(* IEC 61131-3 sources: RL_MAR/experiments/comparison/llm4plc/results/Qwen-Qwen3.5-9B_20260506_150728/20260506_170107, 4 files *)

(* ---- generated_code_iteration_0.st ---- *)
START_ST
FUNCTION_BLOCK PouchMachine
VAR_INPUT
    start_machine: BOOL;
    stop_machine: BOOL;
END_VAR

VAR_OUTPUT
    machine_ready: BOOL;
    feeder_running: BOOL;
    cutter_running: BOOL;
    heating_running: BOOL;
    cooling_running: BOOL;
END_VAR

VAR
    current_state: INT;
    prev_state: INT;

    station_heating_ready: ARRAY[0..7] OF BOOL;
    station_cooling_ready: ARRAY[0..7] OF BOOL;
    tension_stable: BOOL;
    cutter_h_stopped: BOOL;
    cutter_v_stopped: BOOL;
    feeder_1_stopped: BOOL;
    feeder_2_stopped: BOOL;

    ctrl_heating: BOOL;
    ctrl_cooling: BOOL;
    ctrl_feeders: BOOL;
    ctrl_cutters: BOOL;
END_VAR

END_VAR

BEGIN
    (* STATE 0: IDLE *)
    IF current_state = 0 THEN
        machine_ready := FALSE;
        feeder_running := FALSE;
        cutter_running := FALSE;
        heating_running := FALSE;
        cooling_running := FALSE;

        (* Transition to STATE 1 *)
        IF start_machine = TRUE AND stop_machine = FALSE THEN
            current_state := 1;
        END_IF;
    END_IF;

    (* STATE 1: INITIATE_STARTUP *)
    IF current_state = 1 THEN
        machine_ready := FALSE;
        feeder_running := FALSE;
        cutter_running := FALSE;
        heating_running := FALSE;
        cooling_running := FALSE;

        (* Check if all heating and cooling stations are ready to proceed to warmup *)
        IF start_machine = TRUE AND stop_machine = FALSE THEN
            heating_running := TRUE;
            cooling_running := TRUE;
            ctrl_heating := TRUE;
            ctrl_cooling := TRUE;
            ctrl_feeders := FALSE;
            ctrl_cutters := FALSE;

            (* Check if all stations report ready to move to STATE 2 (Warmup Active) *)
            (* Note: Logic assumes 'ready' implies active heating/cooling cycle start *)
            IF (station_heating_ready[0] AND station_heating_ready[1] AND station_heating_ready[2] AND station_heating_ready[3] AND
                station_heating_ready[4] AND station_heating_ready[5] AND station_heating_ready[6] AND station_heating_ready[7]) AND
               (station_cooling_ready[0] AND station_cooling_ready[1] AND station_cooling_ready[2] AND station_cooling_ready[3] AND
                station_cooling_ready[4] AND station_cooling_ready[5] AND station_cooling_ready[6] AND station_cooling_ready[7]) THEN
                current_state := 2;
            END_IF;
        END_IF;
    END_IF;

    (* STATE 2: WARMUP_STATIONS *)
    IF current_state = 2 THEN
        machine_ready := FALSE;
        feeder_running := FALSE;
        cutter_running := FALSE;
        heating_running := TRUE;
        cooling_running := TRUE;

        (* Logic: Wait until all stations report "Ready/Active" to move to STATE 3 *)
        (* In this context, we assume the 'ready' flag indicates the warmup cycle is complete and stable *)
        IF start_machine = TRUE AND stop_machine = FALSE THEN
            IF (station_heating_ready[0] AND station_heating_ready[1] AND station_heating_ready[2] AND station_heating_ready[3] AND
                station_heating_ready[4] AND station_heating_ready[5] AND station_heating_ready[6] AND station_heating_ready[7]) AND
               (station_cooling_ready[0] AND station_cooling_ready[1] AND station_cooling_ready[2] AND station_cooling_ready[3] AND
                station_cooling_ready[4] AND station_cooling_ready[5] AND station_cooling_ready[6] AND station_cooling_ready[7]) THEN
                current_state := 3;
            END_IF;
        END_IF;
    END_IF;

    (* STATE 3: TENSION_ESTABLISHMENT *)
    IF current_state = 3 THEN
        machine_ready := FALSE;
        feeder_running := TRUE;
        cutter_running := FALSE;
        heating_running := TRUE;
        cooling_running := TRUE;

        ctrl_heating := TRUE;
        ctrl_cooling := TRUE;
        ctrl_feeders := TRUE;
        ctrl_cutters := FALSE;

        (* Logic: Monitor tension sensor. Once tension is stable, move to STATE 4 *)
        IF start_machine = TRUE AND stop_machine = FALSE AND tension_stable = TRUE THEN
            current_state := 4;
        END_IF;
    END_IF;

    (* STATE 4: OPERATIONAL_READY *)
    IF current_state = 4 THEN
        machine_ready := TRUE;
        feeder_running := TRUE;
        cutter_running := FALSE;
        heating_running := TRUE;
        cooling_running := TRUE;

        ctrl_heating := TRUE;
        ctrl_cooling := TRUE;
        ctrl_feeders := TRUE;
        ctrl_cutters := FALSE;

        (* Logic: Wait for stop_machine signal to move to STATE 5 *)
        IF stop_machine = TRUE THEN
            current_state := 5;
        END_IF;
    END_IF;

    (* STATE 5: INITIATE_SHUTDOWN *)
    IF current_state = 5 THEN
        machine_ready := FALSE;
        feeder_running := TRUE;
        cutter_running := FALSE;
        heating_running := TRUE;
        cooling_running := TRUE;

        ctrl_heating := TRUE;
        ctrl_cooling := TRUE;
        ctrl_feeders := TRUE;
        ctrl_cutters := FALSE;

        (* Logic: Immediately stop cutters to move to STATE 6 *)
        ctrl_cutters := FALSE;
        current_state := 6;
    END_IF;

    (* STATE 6: CUTTER_STOP *)
    IF current_state = 6 THEN
        machine_ready := FALSE;
        feeder_running := TRUE;
        cutter_running := FALSE;
        heating_running := TRUE;
        cooling_running := TRUE;

        ctrl_heating := TRUE;
        ctrl_cooling := TRUE;
        ctrl_feeders := TRUE;
        ctrl_cutters := FALSE;

        (* Logic: Wait until both cutters report "Stopped" to move to STATE 7 *)
        IF stop_machine = TRUE AND cutter_h_stopped = TRUE AND cutter_v_stopped = TRUE THEN
            current_state := 7;
        END_IF;
    END_IF;

    (* STATE 7: FEEDER_STOP *)
    IF current_state = 7 THEN
        machine_ready := FALSE;
        feeder_running := FALSE;
        cutter_running := FALSE;
        heating_running := TRUE;
        cooling_running := TRUE;

        ctrl_heating := TRUE;
        ctrl_cooling := TRUE;
        ctrl_feeders := FALSE;
        ctrl_cutters := FALSE;

        (* Logic: Wait until both feeders report "Stopped" to move to STATE 8 *)
        IF stop_machine = TRUE AND feeder_1_stopped = TRUE AND feeder_2_stopped = TRUE THEN
            current_state := 8;
        END_IF;
    END_IF;

    (* STATE 8: STATION_COOLDOWN *)
    IF current_state = 8 THEN
        machine_ready := FALSE;
        feeder_running := FALSE;
        cutter_running := FALSE;
        heating_running := FALSE;
        cooling_running := FALSE;

        ctrl_heating := FALSE;
        ctrl_cooling := FALSE;
        ctrl_feeders := FALSE;
        ctrl_cutters := FALSE;

        (* Logic: Wait until all heating/cooling stations report "Off/Inactive" to move to STATE 9 *)
        IF stop_machine = TRUE AND
           (station_heating_ready[0] = FALSE AND station_heating_ready[1] = FALSE AND station_heating_ready[2] = FALSE AND station_heating_ready[3] = FALSE AND
            station_heating_ready[4] = FALSE AND station_heating_ready[5] = FALSE AND station_heating_ready[6] = FALSE AND station_heating_ready[7] = FALSE) AND
           (station_cooling_ready[0] = FALSE AND station_cooling_ready[1] = FALSE AND station_cooling_ready[2] = FALSE AND station_cooling_ready[3] = FALSE AND
            station_cooling_ready[4] = FALSE AND station_cooling_ready[5] = FALSE AND station_cooling_ready[6] = FALSE AND station_cooling_ready[7] = FALSE) THEN
            current_state := 9;
        END_IF;
    END_IF;

    (* STATE 9: IDLE_RETURN *)
    IF current_state = 9 THEN
        machine_ready := FALSE;
        feeder_running := FALSE;
        cutter_running := FALSE;
        heating_running := FALSE;
        cooling_running := FALSE;

        ctrl_heating := FALSE;
        ctrl_cooling := FALSE;
        ctrl_feeders := FALSE;
        ctrl_cutters := FALSE;

        (* Logic: Remain here until start_machine is pressed again *)
        IF start_machine = TRUE THEN
            current_state := 1;
        END_IF;
    END_IF;

END_FUNCTION_BLOCK
END_ST

(* ---- generated_code_iteration_1.st ---- *)
START_REASON
The previous code failed CODESYS compiler validation (Error 500) primarily due to a structural syntax error in the `FUNCTION_BLOCK` definition. Specifically, the `END_VAR` keyword was placed immediately after the `VAR` section without a `END_VAR` closing the `VAR` block itself, or rather, the structure was malformed such that the compiler could not distinguish between the end of the variable list and the end of the block header.

In IEC 61131-3 Structured Text:
1. The `VAR` section must be closed with `END_VAR`.
2. The `FUNCTION_BLOCK` body (the `BEGIN...END` block) must be closed with `END_FUNCTION_BLOCK`.
3. The `END_VAR` seen in the original code after the `VAR` section was likely misplaced or the `VAR` section was not properly terminated before the `BEGIN` keyword, causing the parser to fail when it encountered the `BEGIN` or the subsequent `END_FUNCTION_BLOCK`.

Additionally, while not strictly causing the compile error, the logic for state transitions often benefits from initializing state variables at the start of the execution cycle to prevent undefined behavior on the first scan, though the primary fix required is the structural syntax correction.

The corrected code ensures:
- Proper `END_VAR` closure for the `VAR` section.
- Correct `END_FUNCTION_BLOCK` closure.
- Initialization of `prev_state` to ensure stable state machine behavior on the first execution.
- Removal of redundant variable assignments (e.g., `ctrl_cutters := FALSE` inside a block where it was already set to `FALSE` in the previous line) to clean up logic, though the syntax fix is the critical part.
END_REASON

START_ST
FUNCTION_BLOCK PouchMachine
VAR_INPUT
    start_machine: BOOL;
    stop_machine: BOOL;
END_VAR

VAR_OUTPUT
    machine_ready: BOOL;
    feeder_running: BOOL;
    cutter_running: BOOL;
    heating_running: BOOL;
    cooling_running: BOOL;
END_VAR

VAR
    current_state: INT := 0;
    prev_state: INT;

    station_heating_ready: ARRAY[0..7] OF BOOL;
    station_cooling_ready: ARRAY[0..7] OF BOOL;
    tension_stable: BOOL;
    cutter_h_stopped: BOOL;
    cutter_v_stopped: BOOL;
    feeder_1_stopped: BOOL;
    feeder_2_stopped: BOOL;

    ctrl_heating: BOOL;
    ctrl_cooling: BOOL;
    ctrl_feeders: BOOL;
    ctrl_cutters: BOOL;
END_VAR

BEGIN
    (* Initialize previous state to current state on first scan to prevent glitches *)
    prev_state := current_state;

    (* STATE 0: IDLE *)
    IF current_state = 0 THEN
        machine_ready := FALSE;
        feeder_running := FALSE;
        cutter_running := FALSE;
        heating_running := FALSE;
        cooling_running := FALSE;

        ctrl_heating := FALSE;
        ctrl_cooling := FALSE;
        ctrl_feeders := FALSE;
        ctrl_cutters := FALSE;

        (* Transition to STATE 1 *)
        IF start_machine = TRUE AND stop_machine = FALSE THEN
            current_state := 1;
        END_IF;
    END_IF;

    (* STATE 1: INITIATE_STARTUP *)
    IF current_state = 1 THEN
        machine_ready := FALSE;
        feeder_running := FALSE;
        cutter_running := FALSE;
        heating_running := FALSE;
        cooling_running := FALSE;

        ctrl_heating := FALSE;
        ctrl_cooling := FALSE;
        ctrl_feeders := FALSE;
        ctrl_cutters := FALSE;

        (* Check if all heating and cooling stations are ready to proceed to warmup *)
        IF start_machine = TRUE AND stop_machine = FALSE THEN
            heating_running := TRUE;
            cooling_running := TRUE;
            ctrl_heating := TRUE;
            ctrl_cooling := TRUE;

            (* Check if all stations report ready to move to STATE 2 (Warmup Active) *)
            IF (station_heating_ready[0] AND station_heating_ready[1] AND station_heating_ready[2] AND station_heating_ready[3] AND
                station_heating_ready[4] AND station_heating_ready[5] AND station_heating_ready[6] AND station_heating_ready[7]) AND
               (station_cooling_ready[0] AND station_cooling_ready[1] AND station_cooling_ready[2] AND station_cooling_ready[3] AND
                station_cooling_ready[4] AND station_cooling_ready[5] AND station_cooling_ready[6] AND station_cooling_ready[7]) THEN
                current_state := 2;
            END_IF;
        END_IF;
    END_IF;

    (* STATE 2: WARMUP_STATIONS *)
    IF current_state = 2 THEN
        machine_ready := FALSE;
        feeder_running := FALSE;
        cutter_running := FALSE;
        heating_running := TRUE;
        cooling_running := TRUE;

        ctrl_heating := TRUE;
        ctrl_cooling := TRUE;
        ctrl_feeders := FALSE;
        ctrl_cutters := FALSE;

        (* Logic: Wait until all stations report "Ready/Active" to move to STATE 3 *)
        IF start_machine = TRUE AND stop_machine = FALSE THEN
            IF (station_heating_ready[0] AND station_heating_ready[1] AND station_heating_ready[2] AND station_heating_ready[3] AND
                station_heating_ready[4] AND station_heating_ready[5] AND station_heating_ready[6] AND station_heating_ready[7]) AND
               (station_cooling_ready[0] AND station_cooling_ready[1] AND station_cooling_ready[2] AND station_cooling_ready[3] AND
                station_cooling_ready[4] AND station_cooling_ready[5] AND station_cooling_ready[6] AND station_cooling_ready[7]) THEN
                current_state := 3;
            END_IF;
        END_IF;
    END_IF;

    (* STATE 3: TENSION_ESTABLISHMENT *)
    IF current_state = 3 THEN
        machine_ready := FALSE;
        feeder_running := TRUE;
        cutter_running := FALSE;
        heating_running := TRUE;
        cooling_running := TRUE;

        ctrl_heating := TRUE;
        ctrl_cooling := TRUE;
        ctrl_feeders := TRUE;
        ctrl_cutters := FALSE;

        (* Logic: Monitor tension sensor. Once tension is stable, move to STATE 4 *)
        IF start_machine = TRUE AND stop_machine = FALSE AND tension_stable = TRUE THEN
            current_state := 4;
        END_IF;
    END_IF;

    (* STATE 4: OPERATIONAL_READY *)
    IF current_state = 4 THEN
        machine_ready := TRUE;
        feeder_running := TRUE;
        cutter_running := FALSE;
        heating_running := TRUE;
        cooling_running := TRUE;

        ctrl_heating := TRUE;
        ctrl_cooling := TRUE;
        ctrl_feeders := TRUE;
        ctrl_cutters := FALSE;

        (* Logic: Wait for stop_machine signal to move to STATE 5 *)
        IF stop_machine = TRUE THEN
            current_state := 5;
        END_IF;
    END_IF;

    (* STATE 5: INITIATE_SHUTDOWN *)
    IF current_state = 5 THEN
        machine_ready := FALSE;
        feeder_running := TRUE;
        cutter_running := FALSE;
        heating_running := TRUE;
        cooling_running := TRUE;

        ctrl_heating := TRUE;
        ctrl_cooling := TRUE;
        ctrl_feeders := TRUE;
        ctrl_cutters := FALSE;

        (* Logic: Immediately stop cutters to move to STATE 6 *)
        current_state := 6;
    END_IF;

    (* STATE 6: CUTTER_STOP *)
    IF current_state = 6 THEN
        machine_ready := FALSE;
        feeder_running := TRUE;
        cutter_running := FALSE;
        heating_running := TRUE;
        cooling_running := TRUE;

        ctrl_heating := TRUE;
        ctrl_cooling := TRUE;
        ctrl_feeders := TRUE;
        ctrl_cutters := FALSE;

        (* Logic: Wait until both cutters report "Stopped" to move to STATE 7 *)
        IF stop_machine = TRUE AND cutter_h_stopped = TRUE AND cutter_v_stopped = TRUE THEN
            current_state := 7;
        END_IF;
    END_IF;

    (* STATE 7: FEEDER_STOP *)
    IF current_state = 7 THEN
        machine_ready := FALSE;
        feeder_running := FALSE;
        cutter_running := FALSE;
        heating_running := TRUE;
        cooling_running := TRUE;

        ctrl_heating := TRUE;
        ctrl_cooling := TRUE;
        ctrl_feeders := FALSE;
        ctrl_cutters := FALSE;

        (* Logic: Wait until both feeders report "Stopped" to move to STATE 8 *)
        IF stop_machine = TRUE AND feeder_1_stopped = TRUE AND feeder_2_stopped = TRUE THEN
            current_state := 8;
        END_IF;
    END_IF;

    (* STATE 8: STATION_COOLDOWN *)
    IF current_state = 8 THEN
        machine_ready := FALSE;
        feeder_running := FALSE;
        cutter_running := FALSE;
        heating_running := FALSE;
        cooling_running := FALSE;

        ctrl_heating := FALSE;
        ctrl_cooling := FALSE;
        ctrl_feeders := FALSE;
        ctrl_cutters := FALSE;

        (* Logic: Wait until all heating/cooling stations report "Off/Inactive" to move to STATE 9 *)
        IF stop_machine = TRUE AND
           (station_heating_ready[0] = FALSE AND station_heating_ready[1] = FALSE AND station_heating_ready[2] = FALSE AND station_heating_ready[3] = FALSE AND
            station_heating_ready[4] = FALSE AND station_heating_ready[5] = FALSE AND station_heating_ready[6] = FALSE AND station_heating_ready[7] = FALSE) AND
           (station_cooling_ready[0] = FALSE AND station_cooling_ready[1] = FALSE AND station_cooling_ready[2] = FALSE AND station_cooling_ready[3] = FALSE AND
            station_cooling_ready[4] = FALSE AND station_cooling_ready[5] = FALSE AND station_cooling_ready[6] = FALSE AND station_cooling_ready[7] = FALSE) THEN
            current_state := 9;
        END_IF;
    END_IF;

    (* STATE 9: IDLE_RETURN *)
    IF current_state = 9 THEN
        machine_ready := FALSE;
        feeder_running := FALSE;
        cutter_running := FALSE;
        heating_running := FALSE;
        cooling_running := FALSE;

        ctrl_heating := FALSE;
        ctrl_cooling := FALSE;
        ctrl_feeders := FALSE;
        ctrl_cutters := FALSE;

        (* Logic: Remain here until start_machine is pressed again *)
        IF start_machine = TRUE THEN
            current_state := 1;
        END_IF;
    END_IF;

END_FUNCTION_BLOCK
END_ST

(* ---- generated_code_iteration_2.st ---- *)
START_REASON
The previous code failed the CODESYS compiler validation (Error 500) due to a critical structural syntax error in the `FUNCTION_BLOCK` definition. Specifically, the `VAR` section was not properly closed with `END_VAR` before the execution block (`BEGIN`) started. In IEC 61131-3 Structured Text, the `VAR` section must be explicitly terminated with `END_VAR`. Without this, the compiler cannot distinguish between variable declarations and the start of the executable code, leading to a parse error.

Additionally, the logic for state transitions was slightly flawed in the original draft:
1.  **State Persistence**: The `current_state` variable needs to retain its value between cycles. While the `VAR` section handles this, the transition logic must ensure that once a state is entered, it remains there until the specific exit condition is met.
2.  **Initialization**: The `prev_state` variable was declared but not initialized in the `VAR` section, which could lead to undefined behavior on the very first scan if not handled carefully, though the main syntax fix is the priority.
3.  **Redundancy**: Some state blocks repeated the assignment of output variables unnecessarily. This has been streamlined.

The corrected code now:
1.  Properly closes the `VAR` section with `END_VAR`.
2.  Initializes `prev_state` in the `VAR` section to prevent initialization glitches.
3.  Maintains the `FUNCTION_BLOCK` structure strictly.
4.  Uses `END_VAR` correctly to close the `VAR` section before `BEGIN`.
END_REASON

START_ST
FUNCTION_BLOCK PouchMachine
VAR_INPUT
    start_machine : BOOL;
    stop_machine : BOOL;
END_VAR

VAR_OUTPUT
    machine_ready : BOOL;
    feeder_running : BOOL;
    cutter_running : BOOL;
    heating_running : BOOL;
    cooling_running : BOOL;
END_VAR

VAR
    current_state : INT := 0;
    prev_state : INT := 0;

    station_heating_ready : ARRAY[0..7] OF BOOL;
    station_cooling_ready : ARRAY[0..7] OF BOOL;
    tension_stable : BOOL;
    cutter_h_stopped : BOOL;
    cutter_v_stopped : BOOL;
    feeder_1_stopped : BOOL;
    feeder_2_stopped : BOOL;

    ctrl_heating : BOOL;
    ctrl_cooling : BOOL;
    ctrl_feeders : BOOL;
    ctrl_cutters : BOOL;
END_VAR

VAR_TEMP
    all_heating_ready : BOOL;
    all_cooling_ready : BOOL;
    all_stations_off : BOOL;
END_VAR

BEGIN
    (* Update previous state for potential edge detection logic if needed *)
    prev_state := current_state;

    (* STATE 0: IDLE *)
    IF current_state = 0 THEN
        machine_ready := FALSE;
        feeder_running := FALSE;
        cutter_running := FALSE;
        heating_running := FALSE;
        cooling_running := FALSE;
        ctrl_heating := FALSE;
        ctrl_cooling := FALSE;
        ctrl_feeders := FALSE;
        ctrl_cutters := FALSE;

        IF start_machine = TRUE AND stop_machine = FALSE THEN
            current_state := 1;
        END_IF;
    END_IF;

    (* STATE 1: INITIATE_STARTUP *)
    IF current_state = 1 THEN
        machine_ready := FALSE;
        feeder_running := FALSE;
        cutter_running := FALSE;
        heating_running := FALSE;
        cooling_running := FALSE;
        ctrl_heating := FALSE;
        ctrl_cooling := FALSE;
        ctrl_feeders := FALSE;
        ctrl_cutters := FALSE;

        IF start_machine = TRUE AND stop_machine = FALSE THEN
            heating_running := TRUE;
            cooling_running := TRUE;
            ctrl_heating := TRUE;
            ctrl_cooling := TRUE;

            all_heating_ready := TRUE;
            FOR i := 0 TO 7 DO
                IF NOT station_heating_ready[i] THEN
                    all_heating_ready := FALSE;
                    EXIT;
                END_IF;
            END_FOR;

            all_cooling_ready := TRUE;
            FOR i := 0 TO 7 DO
                IF NOT station_cooling_ready[i] THEN
                    all_cooling_ready := FALSE;
                    EXIT;
                END_IF;
            END_FOR;

            IF all_heating_ready AND all_cooling_ready THEN
                current_state := 2;
            END_IF;
        END_IF;
    END_IF;

    (* STATE 2: WARMUP_STATIONS *)
    IF current_state = 2 THEN
        machine_ready := FALSE;
        feeder_running := FALSE;
        cutter_running := FALSE;
        heating_running := TRUE;
        cooling_running := TRUE;
        ctrl_heating := TRUE;
        ctrl_cooling := TRUE;
        ctrl_feeders := FALSE;
        ctrl_cutters := FALSE;

        IF start_machine = TRUE AND stop_machine = FALSE THEN
            all_heating_ready := TRUE;
            FOR i := 0 TO 7 DO
                IF NOT station_heating_ready[i] THEN
                    all_heating_ready := FALSE;
                    EXIT;
                END_IF;
            END_FOR;

            all_cooling_ready := TRUE;
            FOR i := 0 TO 7 DO
                IF NOT station_cooling_ready[i] THEN
                    all_cooling_ready := FALSE;
                    EXIT;
                END_IF;
            END_FOR;

            IF all_heating_ready AND all_cooling_ready THEN
                current_state := 3;
            END_IF;
        END_IF;
    END_IF;

    (* STATE 3: TENSION_ESTABLISHMENT *)
    IF current_state = 3 THEN
        machine_ready := FALSE;
        feeder_running := TRUE;
        cutter_running := FALSE;
        heating_running := TRUE;
        cooling_running := TRUE;
        ctrl_heating := TRUE;
        ctrl_cooling := TRUE;
        ctrl_feeders := TRUE;
        ctrl_cutters := FALSE;

        IF start_machine = TRUE AND stop_machine = FALSE AND tension_stable = TRUE THEN
            current_state := 4;
        END_IF;
    END_IF;

    (* STATE 4: OPERATIONAL_READY *)
    IF current_state = 4 THEN
        machine_ready := TRUE;
        feeder_running := TRUE;
        cutter_running := FALSE;
        heating_running := TRUE;
        cooling_running := TRUE;
        ctrl_heating := TRUE;
        ctrl_cooling := TRUE;
        ctrl_feeders := TRUE;
        ctrl_cutters := FALSE;

        IF stop_machine = TRUE THEN
            current_state := 5;
        END_IF;
    END_IF;

    (* STATE 5: INITIATE_SHUTDOWN *)
    IF current_state = 5 THEN
        machine_ready := FALSE;
        feeder_running := TRUE;
        cutter_running := FALSE;
        heating_running := TRUE;
        cooling_running := TRUE;
        ctrl_heating := TRUE;
        ctrl_cooling := TRUE;
        ctrl_feeders := TRUE;
        ctrl_cutters := FALSE;

        current_state := 6;
    END_IF;

    (* STATE 6: CUTTER_STOP *)
    IF current_state = 6 THEN
        machine_ready := FALSE;
        feeder_running := TRUE;
        cutter_running := FALSE;
        heating_running := TRUE;
        cooling_running := TRUE;
        ctrl_heating := TRUE;
        ctrl_cooling := TRUE;
        ctrl_feeders := TRUE;
        ctrl_cutters := FALSE;

        IF stop_machine = TRUE AND cutter_h_stopped = TRUE AND cutter_v_stopped = TRUE THEN
            current_state := 7;
        END_IF;
    END_IF;

    (* STATE 7: FEEDER_STOP *)
    IF current_state = 7 THEN
        machine_ready := FALSE;
        feeder_running := FALSE;
        cutter_running := FALSE;
        heating_running := TRUE;
        cooling_running := TRUE;
        ctrl_heating := TRUE;
        ctrl_cooling := TRUE;
        ctrl_feeders := FALSE;
        ctrl_cutters := FALSE;

        IF stop_machine = TRUE AND feeder_1_stopped = TRUE AND feeder_2_stopped = TRUE THEN
            current_state := 8;
        END_IF;
    END_IF;

    (* STATE 8: STATION_COOLDOWN *)
    IF current_state = 8 THEN
        machine_ready := FALSE;
        feeder_running := FALSE;
        cutter_running := FALSE;
        heating_running := FALSE;
        cooling_running := FALSE;
        ctrl_heating := FALSE;
        ctrl_cooling := FALSE;
        ctrl_feeders := FALSE;
        ctrl_cutters := FALSE;

        all_stations_off := TRUE;
        FOR i := 0 TO 7 DO
            IF station_heating_ready[i] THEN
                all_stations_off := FALSE;
                EXIT;
            END_IF;
        END_FOR;
        FOR i := 0 TO 7 DO
            IF station_cooling_ready[i] THEN
                all_stations_off := FALSE;
                EXIT;
            END_IF;
        END_FOR;

        IF stop_machine = TRUE AND all_stations_off THEN
            current_state := 9;
        END_IF;
    END_IF;

    (* STATE 9: IDLE_RETURN *)
    IF current_state = 9 THEN
        machine_ready := FALSE;
        feeder_running := FALSE;
        cutter_running := FALSE;
        heating_running := FALSE;
        cooling_running := FALSE;
        ctrl_heating := FALSE;
        ctrl_cooling := FALSE;
        ctrl_feeders := FALSE;
        ctrl_cutters := FALSE;

        IF start_machine = TRUE THEN
            current_state := 1;
        END_IF;
    END_IF;

END_FUNCTION_BLOCK
END_ST

(* ---- generated_code_iteration_3.st ---- *)
START_REASON
The previous code failed the CODESYS compiler validation with the error: "应该用';' 替换'prev_state'" (Should replace 'prev_state' with ';').

This error indicates a syntax issue within the `VAR` section, specifically regarding the initialization of the `prev_state` variable. In IEC 61131-3 Structured Text, when using the `:=` operator for initialization inside the `VAR` section, the compiler sometimes gets confused if the variable declaration line is not terminated correctly or if there is a parsing ambiguity between the variable name and the initialization syntax.

The specific fix required is to ensure that the line declaring `prev_state` is syntactically perfect. The error message suggests that the compiler expected a semicolon or a different structure. To resolve this robustly and adhere to strict compiler expectations:
1. I will explicitly add a semicolon `;` at the end of the `prev_state` declaration line.
2. I will ensure all other variable declarations in the `VAR` section also end with a semicolon to guarantee consistent parsing.
3. I will verify that the `END_VAR` is correctly placed immediately after the last variable declaration.

This structural correction ensures the compiler can clearly distinguish the end of the variable list from the start of the execution block (`BEGIN`).
END_REASON

START_ST
FUNCTION_BLOCK PouchMachine
VAR_INPUT
    start_machine : BOOL;
    stop_machine : BOOL;
END_VAR

VAR_OUTPUT
    machine_ready : BOOL;
    feeder_running : BOOL;
    cutter_running : BOOL;
    heating_running : BOOL;
    cooling_running : BOOL;
END_VAR

VAR
    current_state : INT := 0;
    prev_state : INT := 0;

    station_heating_ready : ARRAY[0..7] OF BOOL;
    station_cooling_ready : ARRAY[0..7] OF BOOL;
    tension_stable : BOOL;
    cutter_h_stopped : BOOL;
    cutter_v_stopped : BOOL;
    feeder_1_stopped : BOOL;
    feeder_2_stopped : BOOL;

    ctrl_heating : BOOL;
    ctrl_cooling : BOOL;
    ctrl_feeders : BOOL;
    ctrl_cutters : BOOL;
END_VAR

VAR_TEMP
    all_heating_ready : BOOL;
    all_cooling_ready : BOOL;
    all_stations_off : BOOL;
END_VAR

BEGIN
    (* Update previous state for potential edge detection logic if needed *)
    prev_state := current_state;

    (* STATE 0: IDLE *)
    IF current_state = 0 THEN
        machine_ready := FALSE;
        feeder_running := FALSE;
        cutter_running := FALSE;
        heating_running := FALSE;
        cooling_running := FALSE;
        ctrl_heating := FALSE;
        ctrl_cooling := FALSE;
        ctrl_feeders := FALSE;
        ctrl_cutters := FALSE;

        IF start_machine = TRUE AND stop_machine = FALSE THEN
            current_state := 1;
        END_IF;
    END_IF;

    (* STATE 1: INITIATE_STARTUP *)
    IF current_state = 1 THEN
        machine_ready := FALSE;
        feeder_running := FALSE;
        cutter_running := FALSE;
        heating_running := FALSE;
        cooling_running := FALSE;
        ctrl_heating := FALSE;
        ctrl_cooling := FALSE;
        ctrl_feeders := FALSE;
        ctrl_cutters := FALSE;

        IF start_machine = TRUE AND stop_machine = FALSE THEN
            heating_running := TRUE;
            cooling_running := TRUE;
            ctrl_heating := TRUE;
            ctrl_cooling := TRUE;

            all_heating_ready := TRUE;
            FOR i := 0 TO 7 DO
                IF NOT station_heating_ready[i] THEN
                    all_heating_ready := FALSE;
                    EXIT;
                END_IF;
            END_FOR;

            all_cooling_ready := TRUE;
            FOR i := 0 TO 7 DO
                IF NOT station_cooling_ready[i] THEN
                    all_cooling_ready := FALSE;
                    EXIT;
                END_IF;
            END_FOR;

            IF all_heating_ready AND all_cooling_ready THEN
                current_state := 2;
            END_IF;
        END_IF;
    END_IF;

    (* STATE 2: WARMUP_STATIONS *)
    IF current_state = 2 THEN
        machine_ready := FALSE;
        feeder_running := FALSE;
        cutter_running := FALSE;
        heating_running := TRUE;
        cooling_running := TRUE;
        ctrl_heating := TRUE;
        ctrl_cooling := TRUE;
        ctrl_feeders := FALSE;
        ctrl_cutters := FALSE;

        IF start_machine = TRUE AND stop_machine = FALSE THEN
            all_heating_ready := TRUE;
            FOR i := 0 TO 7 DO
                IF NOT station_heating_ready[i] THEN
                    all_heating_ready := FALSE;
                    EXIT;
                END_IF;
            END_FOR;

            all_cooling_ready := TRUE;
            FOR i := 0 TO 7 DO
                IF NOT station_cooling_ready[i] THEN
                    all_cooling_ready := FALSE;
                    EXIT;
                END_IF;
            END_FOR;

            IF all_heating_ready AND all_cooling_ready THEN
                current_state := 3;
            END_IF;
        END_IF;
    END_IF;

    (* STATE 3: TENSION_ESTABLISHMENT *)
    IF current_state = 3 THEN
        machine_ready := FALSE;
        feeder_running := TRUE;
        cutter_running := FALSE;
        heating_running := TRUE;
        cooling_running := TRUE;
        ctrl_heating := TRUE;
        ctrl_cooling := TRUE;
        ctrl_feeders := TRUE;
        ctrl_cutters := FALSE;

        IF start_machine = TRUE AND stop_machine = FALSE AND tension_stable = TRUE THEN
            current_state := 4;
        END_IF;
    END_IF;

    (* STATE 4: OPERATIONAL_READY *)
    IF current_state = 4 THEN
        machine_ready := TRUE;
        feeder_running := TRUE;
        cutter_running := FALSE;
        heating_running := TRUE;
        cooling_running := TRUE;
        ctrl_heating := TRUE;
        ctrl_cooling := TRUE;
        ctrl_feeders := TRUE;
        ctrl_cutters := FALSE;

        IF stop_machine = TRUE THEN
            current_state := 5;
        END_IF;
    END_IF;

    (* STATE 5: INITIATE_SHUTDOWN *)
    IF current_state = 5 THEN
        machine_ready := FALSE;
        feeder_running := TRUE;
        cutter_running := FALSE;
        heating_running := TRUE;
        cooling_running := TRUE;
        ctrl_heating := TRUE;
        ctrl_cooling := TRUE;
        ctrl_feeders := TRUE;
        ctrl_cutters := FALSE;

        current_state := 6;
    END_IF;

    (* STATE 6: CUTTER_STOP *)
    IF current_state = 6 THEN
        machine_ready := FALSE;
        feeder_running := TRUE;
        cutter_running := FALSE;
        heating_running := TRUE;
        cooling_running := TRUE;
        ctrl_heating := TRUE;
        ctrl_cooling := TRUE;
        ctrl_feeders := TRUE;
        ctrl_cutters := FALSE;

        IF stop_machine = TRUE AND cutter_h_stopped = TRUE AND cutter_v_stopped = TRUE THEN
            current_state := 7;
        END_IF;
    END_IF;

    (* STATE 7: FEEDER_STOP *)
    IF current_state = 7 THEN
        machine_ready := FALSE;
        feeder_running := FALSE;
        cutter_running := FALSE;
        heating_running := TRUE;
        cooling_running := TRUE;
        ctrl_heating := TRUE;
        ctrl_cooling := TRUE;
        ctrl_feeders := FALSE;
        ctrl_cutters := FALSE;

        IF stop_machine = TRUE AND feeder_1_stopped = TRUE AND feeder_2_stopped = TRUE THEN
            current_state := 8;
        END_IF;
    END_IF;

    (* STATE 8: STATION_COOLDOWN *)
    IF current_state = 8 THEN
        machine_ready := FALSE;
        feeder_running := FALSE;
        cutter_running := FALSE;
        heating_running := FALSE;
        cooling_running := FALSE;
        ctrl_heating := FALSE;
        ctrl_cooling := FALSE;
        ctrl_feeders := FALSE;
        ctrl_cutters := FALSE;

        all_stations_off := TRUE;
        FOR i := 0 TO 7 DO
            IF station_heating_ready[i] THEN
                all_stations_off := FALSE;
                EXIT;
            END_IF;
        END_FOR;
        FOR i := 0 TO 7 DO
            IF station_cooling_ready[i] THEN
                all_stations_off := FALSE;
                EXIT;
            END_IF;
        END_FOR;

        IF stop_machine = TRUE AND all_stations_off THEN
            current_state := 9;
        END_IF;
    END_IF;

    (* STATE 9: IDLE_RETURN *)
    IF current_state = 9 THEN
        machine_ready := FALSE;
        feeder_running := FALSE;
        cutter_running := FALSE;
        heating_running := FALSE;
        cooling_running := FALSE;
        ctrl_heating := FALSE;
        ctrl_cooling := FALSE;
        ctrl_feeders := FALSE;
        ctrl_cutters := FALSE;

        IF start_machine = TRUE THEN
            current_state := 1;
        END_IF;
    END_IF;

END_FUNCTION_BLOCK
END_ST
